{attribute 'GeneratedUsingTerminal: EJ2522-0000-0022'}
{attribute addProperty BoxType "EJ2522-0000-0022"}
{attribute addProperty Id "StatusAT %I*Status_B83811715"}
{attribute addProperty CRC "3773501672"}
{attribute addProperty Size "5"}
TYPE PTO_Status_Channel_E0EB10E8 EXTENDS InputBase_8311D824 :
STRUCT
	{attribute addProperty Name "Status"}
	Status AT %I* : Status_B8381171;
END_STRUCT
END_TYPE

(* stored: Version 1.2.0.0, ProductVersion 3.1.4024.11
   DUT PTO_Status_Channel_E0EB10E8: Id {86247553-b2dd-4493-829b-f15f9ec7ef3c} *)
